# B&R Automation Studio project Panasonic_LinkaPowerCP2_A2021055 (part 21)

```iecst
			P2_Srobovanie.ServoManipulOsY.Parameters.Velocity:= P2_RemPremenne.P2_ManipSrob_OsY_Rychlost/1000;
			P2_Srobovanie.ServoManipulOsY.Parameters.Position:= P2_RemPremenne.P2_Srob_PozY_OdobratSkrutkyM4; //mm

			IF NOT SC_P2_Srobovanie.Switch1 AND P2_Pracovisko.STAV.SkrutkovackyZasunute THEN
				P2_Srobovanie.ServoManipulOsX.Command.MovePosition:= TRUE;
				P2_Srobovanie.ServoManipulOsY.Command.MovePosition:= TRUE;
				SC_P2_Srobovanie.Switch1:= TRUE;
			END_IF

			IF P2_Srobovanie.ServoManipulOsX.Status.InPosition AND P2_Srobovanie.ServoManipulOsY.Status.InPosition THEN
				P2_Srobovanie.ServoManipulOsX.Command.MovePosition:= FALSE;
				P2_Srobovanie.ServoManipulOsY.Command.MovePosition:= FALSE;
				P2_Srobovanie.STAV.ManipulatorNadPodavacmi:= TRUE;
				SC_P2_Srobovanie.ResetStep:= TRUE;
				SC_P2_Srobovanie.Step:= 242;
			END_IF

		242:
			SC_P2_Srobovanie.StepName:='242 - Automaticky Rezim - model 5H, kontrola skrutky M4 na vystupe podavaca';
			SC_P2_Srobovanie.IdleTime.PT:= T#200ms;
			SC_P2_Srobovanie.AlarmTime.PT:= T#10s;
			SC_P2_Srobovanie.AlarmTime.IN:= TRUE;

			IF P2_Srobovanie.SkrutSet_M4.IN.Podavac_SkrutkaNaVystupe THEN
				SC_P2_Srobovanie.ResetStep:= TRUE;
				SC_P2_Srobovanie.Step:= 244;
			ELSE
				P2_Srobovanie.CMD.PodajSkrutku_M4:= TRUE;
				SC_P2_Srobovanie.ResetStep:= TRUE;
				SC_P2_Srobovanie.Step:= 243;
			END_IF

		243:
			SC_P2_Srobovanie.StepName:='243 - Automaticky Rezim - model 5H, cakam na podanie skrutky M4';
			SC_P2_Srobovanie.IdleTime.PT:= T#200ms;
			SC_P2_Srobovanie.AlarmTime.PT:= T#10s;

			IF P2_Srobovanie.SkrutSet_M4.IN.Podavac_SkrutkaNaVystupe THEN
				SC_P2_Srobovanie.ResetStep:= TRUE;
				SC_P2_Srobovanie.Step:= 242;
			ELSIF P2_Srobovanie.SkrutSet_M4.STAV.ERROR THEN
				P2_Alarmy[237]:= TRUE;
				P2_Pracovisko.STAV.Porucha_ST4:= TRUE;
			END_IF

		244:
			SC_P2_Srobovanie.StepName:='244 - Automaticky Rezim - model 5H,vysunutie skrutkovacky pre odobratie skrutky M4 z podavaca';
			SC_P2_Srobovanie.IdleTime.PT:= T#2s;
			SC_P2_Srobovanie.AlarmTime.PT:= T#10s;

			P2_Srobovanie.ServoManipulOsZ_M4.Parameters.Velocity:= P2_RemPremenne.P2_ManipSrob_OsZ_M4_Rychlost/1000;
			P2_Srobovanie.ServoManipulOsZ_M4.Parameters.Position:= P2_RemPremenne.P2_Srob_PozZ_OdobratSkrutkyM4;

			IF NOT SC_P2_Srobovanie.Switch1 THEN
				P2_Srobovanie.ServoManipulOsZ_M4.Command.MovePosition:= TRUE;
				SC_P2_Srobovanie.Switch1:= TRUE;
			END_IF

			IF P2_Srobovanie.ServoManipulOsZ_M4.Status.InPosition THEN
				P2_Srobovanie.OUT.Skrutkovacka_M4_Prisavanie_OFF:= FALSE;
				P2_Srobovanie.OUT.Skrutkovacka_M4_Prisavanie_ON:= TRUE;
				SC_P2_Srobovanie.AlarmTime.IN:= TRUE;
			END_IF

			IF P2_Srobovanie.ServoManipulOsZ_M4.Status.InPosition AND P2_Srobovanie.IN.Skrutkovacka_M4_Vakum_OK THEN
				P2_Srobovanie.ServoManipulOsZ_M4.Command.MovePosition:= FALSE;
				SC_P2_Srobovanie.ResetStep:= TRUE;
				SC_P2_Srobovanie.Step:= 245;
			ELSIF SC_P2_Srobovanie.AlarmTime.Q THEN
				P2_Srobovanie.ServoManipulOsZ_M4.Command.MovePosition:= FALSE;
				P2_Srobovanie.OUT.Skrutkovacka_M4_Prisavanie_ON:= FALSE;
				P2_Srobovanie.OUT.Skrutkovacka_M4_Prisavanie_OFF:= TRUE;
				P2_Alarmy[237]:= TRUE;
				P2_Srobovanie.COM_OUT.Stav_PoruchaSkrutkovania:= TRUE;
				SC_P2_Srobovanie.ResetStep:= TRUE;
				SC_P2_Srobovanie.Step:= 245;
			END_IF

		245:
			SC_P2_Srobovanie.StepName:='245 - Automaticky Rezim - model 5H,zasunutie skrutkovacky po odobrati skrutky M4 z podavaca';
			SC_P2_Srobovanie.IdleTime.PT:= T#2s;
			SC_P2_Srobovanie.AlarmTime.PT:= T#30s;

			P2_Srobovanie.ServoManipulOsZ_M4.Parameters.Velocity:= P2_RemPremenne.P2_ManipSrob_OsZ_M4_Rychlost/1000;
			P2_Srobovanie.ServoManipulOsZ_M4.Parameters.Position:= 0;

			IF NOT SC_P2_Srobovanie.Switch1 THEN
				P2_Srobovanie.ServoManipulOsZ_M4.Command.MovePosition:= TRUE;
				SC_P2_Srobovanie.Switch1:= TRUE;
			END_IF

			IF EDGEPOS(P2_Srobovanie.ServoManipulOsZ_M4.Status.InPosition) THEN
				P2_Srobovanie.ServoManipulOsZ_M4.Command.MovePosition:= FALSE;
				IF P2_Srobovanie.COM_OUT.Stav_PoruchaSkrutkovania THEN
					P2_Pracovisko.STAV.Porucha_ST4:= TRUE;
				ELSE
					SC_P2_Srobovanie.ResetStep:= TRUE;
					SC_P2_Srobovanie.Step:= 246;
				END_IF
			END_IF

		246:
			SC_P2_Srobovanie.StepName:='246 - Automaticky Rezim - model 5H,priprava skrutky M4';
			SC_P2_Srobovanie.IdleTime.PT:= T#200ms;
			SC_P2_Srobovanie.AlarmTime.PT:= T#30s;

			P2_Srobovanie.CMD.PodajSkrutku_M4:= TRUE;
			SC_P2_Srobovanie.ResetStep:= TRUE;
			SC_P2_Srobovanie.Step:= 250;

		250:
			SC_P2_Srobovanie.StepName:='160 - Automaticky Rezim - model 5H, napolohovanie na poziciu skrutkovania strednej skrutky M4';
			SC_P2_Srobovanie.IdleTime.PT:= T#200ms;
			SC_P2_Srobovanie.AlarmTime.PT:= T#5s;

			P2_Robot.COM_OUT.ManipSrobovania_BezpecnaPozicia:= FALSE;

			IF NOT P2_Srobovanie.Manual THEN
				P2_Srobovanie.ServoManipulOsX.Parameters.Velocity:= P2_RemPremenne.P2_ManipSrob_OsX_Rychlost/1000; // m/s
				P2_Srobovanie.ServoManipulOsY.Parameters.Velocity:= P2_RemPremenne.P2_ManipSrob_OsY_Rychlost/1000; // m/s
			END_IF

			P2_Srobovanie.ServoManipulOsX.Parameters.Position:= P2_RemPremenne.P2_Srob5H_PozX_SkrutkyM4; //mm
			P2_Srobovanie.ServoManipulOsY.Parameters.Position:= P2_RemPremenne.P2_Srob5H_PozY_SkrutkyM4; //mm

			IF NOT SC_P2_Srobovanie.Switch1 AND P2_Pracovisko.STAV.SkrutkovackyZasunute THEN
				P2_Srobovanie.ServoManipulOsX.Command.MovePosition:= TRUE;
				P2_Srobovanie.ServoManipulOsY.Command.MovePosition:= TRUE;
				P2_Srobovanie.STAV.ManipulatorNadPodavacmi:= FALSE;
				SC_P2_Srobovanie.Switch1:= TRUE;
			END_IF

			IF P2_Srobovanie.ServoManipulOsX.Status.InPosition AND P2_Srobovanie.ServoManipulOsY.Status.InPosition THEN
				P2_Srobovanie.ServoManipulOsX.Command.MovePosition:= FALSE;
				P2_Srobovanie.ServoManipulOsY.Command.MovePosition:= FALSE;
				IF P2_Srobovanie.STAV.RR_Polohovanie_BUSY THEN
					P2_Srobovanie.STAV.RR_Polohovanie_BUSY:= FALSE;
					SC_P2_Srobovanie.ResetStep:= TRUE;
					SC_P2_Srobovanie.Step:= 700;
				ELSE
					SC_P2_Srobovanie.ResetStep:= TRUE;
					SC_P2_Srobovanie.Step:= 251;
				END_IF
			END_IF

		251:
			SC_P2_Srobovanie.StepName:='251 - Automaticky Rezim - model 5H, vymazanie vysledkov srobovania';
			SC_P2_Srobovanie.IdleTime.PT:= T#2s;
			SC_P2_Srobovanie.AlarmTime.PT:= T#5s;

			IF NOT SC_P2_Srobovanie.Switch1 THEN
				P2_Srobovanie.Skrutkovacka_M4.RESET_Vysledkov:= TRUE;
				SC_P2_Srobovanie.Switch1:= TRUE;
			END_IF

			IF NOT P2_Srobovanie.Skrutkovacka_M4.Stav_VysledokUtahovania_NG AND NOT P2_Srobovanie.Skrutkovacka_M4.Stav_VysledokUtahovania_OK AND NOT P2_Srobovanie.Skrutkovacka_M4.Stav_UtahovanieUkoncene THEN
				P2_Srobovanie.Skrutkovacka_M4.RESET_Vysledkov:= FALSE;
				SC_P2_Srobovanie.ResetStep:= TRUE;
				SC_P2_Srobovanie.Step:= 252;
			END_IF

		252:
			SC_P2_Srobovanie.StepName:='252 - Automaticky Rezim - model 5H, kontrola skrutkovacky a skrutky M4 v skrutkovacke';
			SC_P2_Srobovanie.IdleTime.PT:= T#2s;
			SC_P2_Srobovanie.AlarmTime.PT:= T#5s;

			IF P2_Srobovanie.IN.Skrutkovacka_M4_Vakum_OK AND P2_Srobovanie.Skrutkovacka_M4.Stav_READY_to_START THEN
				SC_P2_Srobovanie.ResetStep:= TRUE;
				SC_P2_Srobovanie.Step:= 253;
			ELSIF NOT P2_Srobovanie.Skrutkovacka_M4.Stav_READY_to_START THEN
				P2_Alarmy[275]:= TRUE;
				P2_Pracovisko.STAV.Porucha_ST4:= TRUE;
			ELSIF NOT P2_Srobovanie.IN.Skrutkovacka_M4_Vakum_OK THEN
				P2_Alarmy[237]:= TRUE;
				P2_Pracovisko.STAV.Porucha_ST4:= TRUE;
			END_IF

		253:
			SC_P2_Srobovanie.StepName:='253 - Automaticky Rezim - model 5H, vysunutie skrutkovacky M4 na poziciu pred skrutkovanim a spustenie skrutkovania';
			SC_P2_Srobovanie.IdleTime.PT:= T#500ms;
			SC_P2_Srobovanie.AlarmTime.PT:= T#10s;

			P2_Srobovanie.ServoManipulOsZ_M4.Parameters.Velocity:= P2_RemPremenne.P2_ManipSrob_OsZ_M4_Rychlost/1000;
			P2_Srobovanie.ServoManipulOsZ_M4.Parameters.Position:= 70;

			IF NOT SC_P2_Srobovanie.Switch1 THEN
				P2_Srobovanie.ServoManipulOsZ_M4.Command.MovePosition:= TRUE;
				P2_Srobovanie.Skrutkovacka_M4.START_Utahovania:= TRUE;
				P2_StoperSrobovania.STAV.VyrobaZacala:= TRUE;
				SC_P2_Srobovanie.Switch1:= TRUE;
			END_IF

			IF EDGEPOS(P2_Srobovanie.ServoManipulOsZ_M4.Status.InPosition) THEN
				P2_Srobovanie.ServoManipulOsZ_M4.Command.MovePosition:= FALSE;
				SC_P2_Srobovanie.ResetStep:= TRUE;
				SC_P2_Srobovanie.Step:= 254;
			END_IF

		254:
			SC_P2_Srobovanie.StepName:='254 - Automaticky Rezim - model 5H, prepnutie vysunutie skrutkovacky M4 na momentovy pohyb';
			SC_P2_Srobovanie.IdleTime.PT:= T#500ms;
			SC_P2_Srobovanie.AlarmTime.PT:= T#10s;
			SC_P2_Srobovanie.IdleTime.IN:= TRUE;

			P2_Srobovanie.ServoManipulOsZ_M4.Parameters.Velocity:= P2_RemPremenne.P2_Srob5H_Rychl_SkrutkyM4/1000;
			P2_Srobovanie.ServoManipulOsZ_M4.Parameters.Torque:= P2_RemPremenne.P2_Srob5H_Mom_SkrutkyM4;
			P2_Srobovanie.ServoManipulOsZ_M4.Parameters.Position:= 100;

			IF NOT SC_P2_Srobovanie.Switch1 THEN
				P2_Srobovanie.ServoManipulOsZ_M4.Command.MovePosition:= TRUE;
				SC_P2_Srobovanie.Switch1:= TRUE;
			END_IF

			IF EDGEPOS(P2_Srobovanie.ServoManipulOsZ_M4.Status.InTorque) THEN
				SC_P2_Srobovanie.ResetStep:= TRUE;
				SC_P2_Srobovanie.Step:= 255;
			END_IF

		255:
			SC_P2_Srobovanie.StepName:='255 - Automaticky Rezim - model 45F, cakam na ukoncenie skrutkovania skrutkovacky M4';
			SC_P2_Srobovanie.IdleTime.PT:= T#30s;
			SC_P2_Srobovanie.AlarmTime.PT:= T#10s;
			SC_P2_Srobovanie.IdleTime.IN:= TRUE;
			SC_P2_Srobovanie.AlarmTime.IN:= TRUE;

			IF P2_Srobovanie.Skrutkovacka_M4.Stav_UtahovanieUkoncene THEN
				P2_Srobovanie.Skrutkovacka_M4.START_Utahovania:= FALSE;
				P2_Srobovanie.ServoManipulOsZ_M4.Command.MovePosition:= FALSE;
				CasSrobovania:= TIME_TO_REAL(SC_P2_Srobovanie.IdleTime.ET);
				Reports.Skrutkovacky.VyskaSkrutkovania.P2_StrednaSkrutkaM4:= REAL_TO_STRING(P2_Srobovanie.ServoManipulOsZ_M4.Status.ActPosition);
				Reports.Skrutkovacky.CasSkrutkovania.P2_StrednaSkrutkaM4:= REAL_TO_STRING(CasSrobovania/1000);
				SC_P2_Srobovanie.ResetStep:= TRUE;
				SC_P2_Srobovanie.Step:= 256;
			ELSIF SC_P2_Srobovanie.AlarmTime.Q THEN
				P2_Alarmy[272]:= TRUE;
				CasSrobovania:= TIME_TO_REAL(SC_P2_Srobovanie.IdleTime.ET);
				Reports.Skrutkovacky.VyskaSkrutkovania.P2_StrednaSkrutkaM4:= REAL_TO_STRING(P2_Srobovanie.ServoManipulOsZ_M4.Status.ActPosition);
				Reports.Skrutkovacky.CasSkrutkovania.P2_StrednaSkrutkaM4:= REAL_TO_STRING(CasSrobovania/1000);
				P2_Srobovanie.Skrutkovacka_M4.START_Utahovania:= FALSE;
				P2_Srobovanie.COM_OUT.Stav_PoruchaSkrutkovania:= TRUE;
				P2_Srobovanie.ServoManipulOsZ_M4.Command.MovePosition:= FALSE;
				SC_P2_Srobovanie.ResetStep:= TRUE;
				SC_P2_Srobovanie.Step:= 256;
			END_IF

		256:
			SC_P2_Srobovanie.StepName:='256 - Automaticky Rezim - model 5H, zasunutie skrutkovacky M4 a vypnutie prisavania skrutky';
			SC_P2_Srobovanie.IdleTime.PT:= T#200ms;
			SC_P2_Srobovanie.AlarmTime.PT:= T#5s;

			P2_Srobovanie.ServoManipulOsZ_M4.Parameters.Velocity:= P2_RemPremenne.P2_ManipSrob_OsZ_M4_Rychlost;
			P2_Srobovanie.ServoManipulOsZ_M4.Parameters.Torque:= 1.0;
			P2_Srobovanie.ServoManipulOsZ_M4.Parameters.Position:= 0;

			IF NOT SC_P2_Srobovanie.Switch1 THEN
				P2_Srobovanie.ServoManipulOsZ_M4.Command.MovePosition:= TRUE;
				P2_Srobovanie.OUT.Skrutkovacka_M4_Prisavanie_ON:= FALSE;
				P2_Srobovanie.OUT.Skrutkovacka_M4_Prisavanie_OFF:= TRUE;
				SC_P2_Srobovanie.Switch1:= TRUE;
			END_IF

			IF EDGEPOS(P2_Srobovanie.ServoManipulOsZ_M4.Status.InPosition) THEN
				P2_Srobovanie.ServoManipulOsZ_M4.Command.MovePosition:= FALSE;
				SC_P2_Srobovanie.ResetStep:= TRUE;
				SC_P2_Srobovanie.Step:= 257;
			END_IF

		257:
			SC_P2_Srobovanie.StepName:='257 - Automaticky Rezim - model 5H, kontrola vysledkov skrutkovania strednej skrutky M4';
			SC_P2_Srobovanie.IdleTime.PT:= T#200ms;
			SC_P2_Srobovanie.AlarmTime.PT:= T#5s;

			IF P2_Srobovanie.COM_OUT.Stav_PoruchaSkrutkovania THEN
				P2_Srobovanie.STAV.Vysledok_Srobovania:= 'NG';
				P2_Srobovanie.COM_OUT.Stav_SkrutkovanieUkoncene:= TRUE;
				SC_P2_Srobovanie.ResetStep:= TRUE;
				SC_P2_Srobovanie.Step:= 258;
			ELSIF P2_Srobovanie.Skrutkovacka_M4.Stav_VysledokUtahovania_OK THEN
				P2_Srobovanie.STAV.Vysledok_Srobovania:= 'OK';
				P2_Srobovanie.COM_OUT.Stav_SkrutkovanieUkoncene:= TRUE;
				SC_P2_Srobovanie.ResetStep:= TRUE;
				SC_P2_Srobovanie.Step:= 258;
			ELSIF P2_Srobovanie.Skrutkovacka_M4.Stav_VysledokUtahovania_NG THEN
				P2_Srobovanie.STAV.Vysledok_Srobovania:= 'NG';
				P2_Srobovanie.COM_OUT.Stav_SkrutkovanieUkoncene:= TRUE;
				SC_P2_Srobovanie.ResetStep:= TRUE;
				SC_P2_Srobovanie.Step:= 258;
			END_IF

		258:
			SC_P2_Srobovanie.StepName:='258 - Automaticky Rezim - model 5H, cakam na zrusenie signalu zaskrutkuj strednu skrutku M4';
			SC_P2_Srobovanie.IdleTime.PT:= T#200ms;
			SC_P2_Srobovanie.AlarmTime.PT:= T#5s;

			IF NOT P2_Srobovanie.COM_IN.Model5H_ZaskrutkujStrednuM4 THEN
				P2_Srobovanie.COM_OUT.Stav_SkrutkovanieUkoncene:= FALSE;
				SC_P2_Srobovanie.ResetStep:= TRUE;
				SC_P2_Srobovanie.Step:= 100;
			END_IF

			//Presun manipulátora do pozície VPRED//

		400:
			SC_P2_Srobovanie.StepName:='400 - Automaticky Rezim - napolohovanie manipulatora na prednu poziciu ';
			SC_P2_Srobovanie.IdleTime.PT:= T#200ms;
			SC_P2_Srobovanie.AlarmTime.PT:= T#5s;

			P2_Robot.COM_OUT.ManipSrobovania_BezpecnaPozicia:= FALSE;

			P2_Srobovanie.ServoManipulOsX.Parameters.Velocity:= P2_RemPremenne.P2_ManipSrob_OsX_Rychlost/1000; // m/s
			P2_Srobovanie.ServoManipulOsX.Parameters.Position:= 12.5; //mm

			P2_Srobovanie.ServoManipulOsY.Parameters.Velocity:= P2_RemPremenne.P2_ManipSrob_OsY_Rychlost/1000; // m/s
			P2_Srobovanie.ServoManipulOsY.Parameters.Position:= 375; //mm

			IF NOT SC_P2_Srobovanie.Switch1 AND P2_Pracovisko.STAV.SkrutkovackyZasunute THEN
				P2_Srobovanie.ServoManipulOsY.Command.MovePosition:= TRUE;
				SC_P2_Srobovanie.Switch1:= TRUE;
			END_IF

			IF P2_Srobovanie.ServoManipulOsY.Status.ActPosition > 280 THEN
				P2_Srobovanie.ServoManipulOsX.Command.MovePosition:= TRUE;
			END_IF

			IF P2_Srobovanie.ServoManipulOsX.Status.InPosition AND P2_Srobovanie.ServoManipulOsY.Status.InPosition THEN
				P2_Srobovanie.ServoManipulOsX.Command.MovePosition:= FALSE;
				P2_Srobovanie.ServoManipulOsY.Command.MovePosition:= FALSE;
				P2_Srobovanie.COM_OUT.Stav_PresunManipulUkonceny:= TRUE;
				SC_P2_Srobovanie.ResetStep:= TRUE;
				SC_P2_Srobovanie.Step:= 402;
			END_IF

		402:
			SC_P2_Srobovanie.StepName:='402 - Automaticky Rezim - cakam na zrusenie signalu presun manipulatora vpred';
			SC_P2_Srobovanie.IdleTime.PT:= T#200ms;
			SC_P2_Srobovanie.AlarmTime.PT:= T#5s;

			IF NOT P2_Srobovanie.COM_IN.PresunManipulatora_VPRED THEN
				P2_Srobovanie.COM_OUT.Stav_PresunManipulUkonceny:= FALSE;
				SC_P2_Srobovanie.ResetStep:= TRUE;
				SC_P2_Srobovanie.Step:= 100;
			END_IF

			//Presun manipulátora do pozície VZAD//

		420:
			SC_P2_Srobovanie.StepName:='420 - Automaticky Rezim - napolohovanie manipulatora na zadnu poziciu ';
			SC_P2_Srobovanie.IdleTime.PT:= T#200ms;
			SC_P2_Srobovanie.AlarmTime.PT:= T#5s;

			P2_Robot.COM_OUT.ManipSrobovania_BezpecnaPozicia:= FALSE;

			P2_Srobovanie.ServoManipulOsX.Parameters.Velocity:= P2_RemPremenne.P2_ManipSrob_OsX_Rychlost/1000; // m/s
			P2_Srobovanie.ServoManipulOsX.Parameters.Position:= 12.5; //mm

			P2_Srobovanie.ServoManipulOsY.Parameters.Velocity:= P2_RemPremenne.P2_ManipSrob_OsY_Rychlost/1000; // m/s
			P2_Srobovanie.ServoManipulOsY.Parameters.Position:= 4.5; //mm

			IF NOT SC_P2_Srobovanie.Switch1 AND P2_Pracovisko.STAV.SkrutkovackyZasunute THEN
				P2_Srobovanie.ServoManipulOsX.Command.MovePosition:= TRUE;
				P2_Srobovanie.ServoManipulOsY.Command.MovePosition:= TRUE;
				SC_P2_Srobovanie.Switch1:= TRUE;
			END_IF

			IF P2_Srobovanie.ServoManipulOsX.Status.InPosition AND P2_Srobovanie.ServoManipulOsY.Status.InPosition THEN
				P2_Srobovanie.ServoManipulOsX.Command.MovePosition:= FALSE;
				P2_Srobovanie.ServoManipulOsY.Command.MovePosition:= FALSE;
				P2_Srobovanie.COM_OUT.Stav_PresunManipulUkonceny:= TRUE;
				SC_P2_Srobovanie.ResetStep:= TRUE;
				SC_P2_Srobovanie.Step:= 422;
			END_IF

		422:
			SC_P2_Srobovanie.StepName:='422 - Automaticky Rezim - cakam na zrusenie signalu presun manipulatora vzad';
			SC_P2_Srobovanie.IdleTime.PT:= T#200ms;
			SC_P2_Srobovanie.AlarmTime.PT:= T#5s;

			IF NOT P2_Srobovanie.COM_IN.PresunManipulatora_VZAD THEN
				P2_Srobovanie.COM_OUT.Stav_PresunManipulUkonceny:= FALSE;
				SC_P2_Srobovanie.ResetStep:= TRUE;
				SC_P2_Srobovanie.Step:= 100;
			END_IF

			//Odobratie skrutky M4//
		440:
			SC_P2_Srobovanie.StepName:='440 - Automaticky Rezim - odobratie skrtuky M4, napolohovanie zadnej skrutkovacky M4 na poziciu odobratia skrutky M4 z podavaca';
			SC_P2_Srobovanie.IdleTime.PT:= T#200ms;
			SC_P2_Srobovanie.AlarmTime.PT:= T#5s;

			P2_Robot.COM_OUT.ManipSrobovania_BezpecnaPozicia:= FALSE;

			IF NOT P2_Srobovanie.Manual THEN
				P2_Srobovanie.ServoManipulOsX.Parameters.Velocity:= P2_RemPremenne.P2_ManipSrob_OsX_Rychlost/1000; // m/s
				P2_Srobovanie.ServoManipulOsY.Parameters.Velocity:= P2_RemPremenne.P2_ManipSrob_OsY_Rychlost/1000; // m/s
			END_IF

			P2_Srobovanie.ServoManipulOsX.Parameters.Position:= P2_RemPremenne.P2_Srob_PozX_OdobratSkrutkyM4; //mm
			P2_Srobovanie.ServoManipulOsY.Parameters.Position:= P2_RemPremenne.P2_Srob_PozY_OdobratSkrutkyM4; //mm

			IF NOT SC_P2_Srobovanie.Switch1 AND P2_Pracovisko.STAV.SkrutkovackyZasunute THEN
				P2_Srobovanie.ServoManipulOsX.Command.MovePosition:= TRUE;
				P2_Srobovanie.ServoManipulOsY.Command.MovePosition:= TRUE;
				SC_P2_Srobovanie.Switch1:= TRUE;
			END_IF

			IF P2_Srobovanie.ServoManipulOsX.Status.InPosition AND P2_Srobovanie.ServoManipulOsY.Status.InPosition THEN
				P2_Srobovanie.ServoManipulOsX.Command.MovePosition:= FALSE;
				P2_Srobovanie.ServoManipulOsY.Command.MovePosition:= FALSE;
				P2_Srobovanie.STAV.ManipulatorNadPodavacmi:= TRUE;
				IF P2_Srobovanie.STAV.RR_Polohovanie_BUSY THEN
					P2_Srobovanie.STAV.RR_Polohovanie_BUSY:= FALSE;
					SC_P2_Srobovanie.ResetStep:= TRUE;
					SC_P2_Srobovanie.Step:= 700;
				ELSE
					SC_P2_Srobovanie.ResetStep:= TRUE;
					SC_P2_Srobovanie.Step:= 442;
				END_IF
			END_IF

		442:
			SC_P2_Srobovanie.StepName:='442 - Automaticky Rezim - odobratie skrutky M4, kontrola skrutky M4 na vystupe podavaca';
			SC_P2_Srobovanie.IdleTime.PT:= T#200ms;
			SC_P2_Srobovanie.AlarmTime.PT:= T#10s;
			SC_P2_Srobovanie.AlarmTime.IN:= TRUE;

			IF P2_Srobovanie.IN.Skrutkovacka_M4_Vakum_OK THEN
				SC_P2_Srobovanie.ResetStep:= TRUE;
				SC_P2_Srobovanie.Step:= 450;
			ELSIF P2_Srobovanie.SkrutSet_M4.IN.Podavac_SkrutkaNaVystupe THEN
				SC_P2_Srobovanie.ResetStep:= TRUE;
				SC_P2_Srobovanie.Step:= 447;
			ELSIF NOT P2_Srobovanie.SkrutSet_M4.IN.Podavac_SkrutkaNaVystupe THEN
				P2_Srobovanie.CMD.PodajSkrutku_M4:= TRUE;
				SC_P2_Srobovanie.ResetStep:= TRUE;
				SC_P2_Srobovanie.Step:= 445;
			END_IF

		445:
			SC_P2_Srobovanie.StepName:='445 - Automaticky Rezim - odobratie skrutky M4, cakam na podanie skrutky M4';
			SC_P2_Srobovanie.IdleTime.PT:= T#200ms;
			SC_P2_Srobovanie.AlarmTime.PT:= T#10s;

			IF P2_Srobovanie.SkrutSet_M4.IN.Podavac_SkrutkaNaVystupe THEN
				SC_P2_Srobovanie.ResetStep:= TRUE;
				SC_P2_Srobovanie.Step:= 442;
			ELSIF P2_Srobovanie.SkrutSet_M4.STAV.ERROR THEN
				P2_Alarmy[237]:= TRUE;
				P2_Pracovisko.STAV.Porucha_ST4:= TRUE;
			END_IF

		447:
			SC_P2_Srobovanie.StepName:='447 - Automaticky Rezim - odobratie skrutky M4,vysunutie skrutkovacky pre odobratie skrutky M4 z podavaca';
			SC_P2_Srobovanie.IdleTime.PT:= T#2s;
			SC_P2_Srobovanie.AlarmTime.PT:= T#10s;

			P2_Srobovanie.ServoManipulOsZ_M4.Parameters.Velocity:= P2_RemPremenne.P2_ManipSrob_OsZ_M4_Rychlost/1000;
			P2_Srobovanie.ServoManipulOsZ_M4.Parameters.Position:= P2_RemPremenne.P2_Srob_PozZ_OdobratSkrutkyM4;

			IF NOT SC_P2_Srobovanie.Switch1 THEN
				P2_Srobovanie.ServoManipulOsZ_M4.Command.MovePosition:= TRUE;
				SC_P2_Srobovanie.Switch1:= TRUE;
			END_IF

			IF P2_Srobovanie.ServoManipulOsZ_M4.Status.InPosition THEN
				P2_Srobovanie.OUT.Skrutkovacka_M4_Prisavanie_OFF:= FALSE;
				P2_Srobovanie.OUT.Skrutkovacka_M4_Prisavanie_ON:= TRUE;
				SC_P2_Srobovanie.AlarmTime.IN:= TRUE;
			END_IF

			IF P2_Srobovanie.ServoManipulOsZ_M4.Status.InPosition AND P2_Srobovanie.IN.Skrutkovacka_M4_Vakum_OK THEN
				P2_Srobovanie.ServoManipulOsZ_M4.Command.MovePosition:= FALSE;
				SC_P2_Srobovanie.ResetStep:= TRUE;
				SC_P2_Srobovanie.Step:= 448;
			ELSIF SC_P2_Srobovanie.AlarmTime.Q THEN
				P2_Srobovanie.ServoManipulOsZ_M4.Command.MovePosition:= FALSE;
				P2_Srobovanie.OUT.Skrutkovacka_M4_Prisavanie_ON:= FALSE;
				P2_Srobovanie.OUT.Skrutkovacka_M4_Prisavanie_OFF:= TRUE;
				P2_Alarmy[237]:= TRUE;
				P2_Srobovanie.COM_OUT.Stav_PoruchaSkrutkovania:= TRUE;
				SC_P2_Srobovanie.ResetStep:= TRUE;
				SC_P2_Srobovanie.Step:= 448;
			END_IF

		448:
			SC_P2_Srobovanie.StepName:='448 - Automaticky Rezim - odobratie skrutky M4,zasunutie skrutkovacky po odobrati skrutky M4 z podavaca';
			SC_P2_Srobovanie.IdleTime.PT:= T#2s;
			SC_P2_Srobovanie.AlarmTime.PT:= T#30s;

			P2_Srobovanie.ServoManipulOsZ_M4.Parameters.Velocity:= P2_RemPremenne.P2_ManipSrob_OsZ_M4_Rychlost/1000;
			P2_Srobovanie.ServoManipulOsZ_M4.Parameters.Position:= 0;

			IF NOT SC_P2_Srobovanie.Switch1 THEN
				P2_Srobovanie.ServoManipulOsZ_M4.Command.MovePosition:= TRUE;
				SC_P2_Srobovanie.Switch1:= TRUE;
			END_IF

			IF EDGEPOS(P2_Srobovanie.ServoManipulOsZ_M4.Status.InPosition) THEN
				P2_Srobovanie.ServoManipulOsZ_M4.Command.MovePosition:= FALSE;
				IF P2_Srobovanie.COM_OUT.Stav_PoruchaSkrutkovania THEN
					P2_Pracovisko.STAV.Porucha_ST4:= TRUE;
				ELSE
					SC_P2_Srobovanie.ResetStep:= TRUE;
					SC_P2_Srobovanie.Step:= 450;
				END_IF
			END_IF

		450:
			SC_P2_Srobovanie.StepName:='450 - Automaticky Rezim - odobratie skrutky M4,priprava skrutky M4';
			SC_P2_Srobovanie.IdleTime.PT:= T#200ms;
			SC_P2_Srobovanie.AlarmTime.PT:= T#30s;

			P2_Srobovanie.CMD.PodajSkrutku_M4:= TRUE;
			SC_P2_Srobovanie.ResetStep:= TRUE;
			SC_P2_Srobovanie.Step:= 455;

		455:
			SC_P2_Srobovanie.StepName:='455 - Automaticky Rezim - odobratie skrutky M4, cakam na zrusenie signalu odober skrutku M4';
			SC_P2_Srobovanie.IdleTime.PT:= T#200ms;
			SC_P2_Srobovanie.AlarmTime.PT:= T#5s;

			P2_Srobovanie.COM_OUT.Stav_SkrutkovanieUkoncene:= TRUE;

			IF NOT P2_Srobovanie.COM_IN.OdoberSkrutku_M4 THEN
				P2_Srobovanie.COM_OUT.Stav_SkrutkovanieUkoncene:= FALSE;
				P2_Srobovanie.STAV.ManipulatorNadPodavacmi:= FALSE;
				SC_P2_Srobovanie.ResetStep:= TRUE;
				SC_P2_Srobovanie.Step:= 100;
			END_IF

			//*********************************************************Čistenie skrutkovačiek*****************************************************************************//

			//Čistenie skrutkovačky M5//
		500:
			SC_P2_Srobovanie.StepName:='500 - Automaticky Rezim - cistenie skrutkovacky M5,kontrola zrusenia stavu serva v pozicii';
			SC_P2_Srobovanie.IdleTime.PT:= T#300ms;
			SC_P2_Srobovanie.AlarmTime.PT:= T#5s;

			P2_Srobovanie.STAV.CistenieSkrutkovackyM5_BUSY:= TRUE;
			P2_Srobovanie.STAV.SkrutkaM5_READY:= FALSE;

			IF NOT P2_Srobovanie.ServoManipulOsX.Status.InPosition AND NOT P2_Srobovanie.ServoManipulOsY.Status.InPosition THEN
				SC_P2_Srobovanie.ResetStep:= TRUE;
				SC_P2_Srobovanie.Step:= 501;
			END_IF

		501:
			SC_P2_Srobovanie.StepName:='501 - Automaticky Rezim - cistenie skrutkovacky M5,presun na poziciu zahodenia skrutky';
			SC_P2_Srobovanie.IdleTime.PT:= T#300ms;
			SC_P2_Srobovanie.AlarmTime.PT:= T#5s;

			P2_Robot.COM_OUT.ManipSrobovania_BezpecnaPozicia:= FALSE;

			IF NOT P2_Srobovanie.Manual THEN
				P2_Srobovanie.ServoManipulOsX.Parameters.Velocity:= P2_RemPremenne.P2_ManipSrob_OsX_Rychlost/1000; // m/s
				P2_Srobovanie.ServoManipulOsY.Parameters.Velocity:= P2_RemPremenne.P2_ManipSrob_OsY_Rychlost/1000; // m/s
			END_IF

			P2_Srobovanie.ServoManipulOsX.Parameters.Position:= 35; //mm
			P2_Srobovanie.ServoManipulOsY.Parameters.Position:= 85; //mm

			IF NOT SC_P2_Srobovanie.Switch1 AND P2_Pracovisko.STAV.SkrutkovackyZasunute THEN
				P2_Srobovanie.ServoManipulOsX.Command.MovePosition:= TRUE;
				P2_Srobovanie.ServoManipulOsY.Command.MovePosition:= TRUE;
				SC_P2_Srobovanie.Switch1:= TRUE;
			END_IF

			IF P2_Srobovanie.ServoManipulOsX.Status.InPosition AND P2_Srobovanie.ServoManipulOsY.Status.InPosition THEN
				P2_Srobovanie.ServoManipulOsX.Command.MovePosition:= FALSE;
				P2_Srobovanie.ServoManipulOsY.Command.MovePosition:= FALSE;
				SC_P2_Srobovanie.ResetStep:= TRUE;
				SC_P2_Srobovanie.Step:= 502;
			END_IF

		502:
			SC_P2_Srobovanie.StepName:='502 - Automaticky Rezim - cistenie skrutkovacky M5,vysunutie skrutkovacky M5';
			SC_P2_Srobovanie.IdleTime.PT:= T#1s;
			SC_P2_Srobovanie.AlarmTime.PT:= T#2s;

			IF NOT SC_P2_Srobovanie.Switch1 THEN
				P2_Srobovanie.OUT.Skrutkovacka_M5_Prisavanie_ON:= TRUE;
				P2_Srobovanie.OUT.Skrutkovacku_M5_VYSUN:= TRUE;
				SC_P2_Srobovanie.IdleTime.IN:= TRUE;
				SC_P2_Srobovanie.Switch1:= TRUE;
			END_IF

			IF SC_P2_Srobovanie.IdleTime.Q THEN
				P2_Srobovanie.OUT.Skrutkovacka_M5_Prisavanie_ON:= FALSE;
				SC_P2_Srobovanie.AlarmTime.IN:= TRUE;
			END_IF

			IF SC_P2_Srobovanie.AlarmTime.Q THEN
				P2_Srobovanie.OUT.Skrutkovacku_M5_VYSUN:= FALSE;
				SC_P2_Srobovanie.ResetStep:= TRUE;
				SC_P2_Srobovanie.Step:= 505;
			END_IF

		505:
			SC_P2_Srobovanie.StepName:='505 - Automaticky Rezim - cistenie skrutkovacky M5,nabitie skrutky do skrutkovacky M5';
			SC_P2_Srobovanie.IdleTime.PT:= T#2s;
			SC_P2_Srobovanie.AlarmTime.PT:= T#30s;

			IF NOT SC_P2_Srobovanie.Switch1 AND P2_Srobovanie.IN.Skrutkovacka_M5_ZASUNUTA THEN
				IF P2_Srobovanie.Manual THEN
					P2_Srobovanie.CMD.RR_SkrutSetM5_PodajSkrutku:= TRUE;
				ELSE
					P2_Srobovanie.CMD.PodajSkrutku_M5:= TRUE;
				END_IF
				SC_P2_Srobovanie.Switch1:= TRUE;
			END_IF

			IF P2_Srobovanie.STAV.SkrutkaM5_READY THEN
				P2_Srobovanie.STAV.CistenieSkrutkovackyM5_BUSY:= FALSE;
				SC_P2_Srobovanie.ResetStep:= TRUE;
				SC_P2_Srobovanie.Step:= FazaNavratu;
			ELSIF P2_Srobovanie.SkrutSet_M5.Error.ErrorBit THEN
				P2_Alarmy[238]:= TRUE;
				P2_Pracovisko.STAV.Porucha_ST4:= TRUE;
			END_IF

			//Čistenie skrutkovačky M4//
		520:
			SC_P2_Srobovanie.StepName:='520 - Automaticky Rezim - cistenie skrutkovacky M4,kontrola zrusenia stavu serva v pozicii';
			SC_P2_Srobovanie.IdleTime.PT:= T#300ms;
			SC_P2_Srobovanie.AlarmTime.PT:= T#5s;

			IF NOT P2_Srobovanie.ServoManipulOsX.Status.InPosition AND NOT P2_Srobovanie.ServoManipulOsY.Status.InPosition THEN
				SC_P2_Srobovanie.ResetStep:= TRUE;
				SC_P2_Srobovanie.Step:= 521;
			END_IF

		521:
			SC_P2_Srobovanie.StepName:='521 - Automaticky Rezim - cistenie skrutkovacky M4,presun manipulatora na poziciu zahodenia skrutky M4';
			SC_P2_Srobovanie.IdleTime.PT:= T#300ms;
			SC_P2_Srobovanie.AlarmTime.PT:= T#5s;

			P2_Robot.COM_OUT.ManipSrobovania_BezpecnaPozicia:= FALSE;

			IF NOT P2_Srobovanie.Manual THEN
				P2_Srobovanie.ServoManipulOsX.Parameters.Velocity:= P2_RemPremenne.P2_ManipSrob_OsX_Rychlost/1000; // m/s
				P2_Srobovanie.ServoManipulOsY.Parameters.Velocity:= P2_RemPremenne.P2_ManipSrob_OsY_Rychlost/1000; // m/s
			END_IF

			P2_Srobovanie.ServoManipulOsX.Parameters.Position:= 23; //mm
			P2_Srobovanie.ServoManipulOsY.Parameters.Position:= 150; //mm

			IF NOT SC_P2_Srobovanie.Switch1 AND P2_Pracovisko.STAV.SkrutkovackyZasunute THEN
				P2_Srobovanie.ServoManipulOsX.Command.MovePosition:= TRUE;
				P2_Srobovanie.ServoManipulOsY.Command.MovePosition:= TRUE;
				SC_P2_Srobovanie.Switch1:= TRUE;
			END_IF

			IF P2_Srobovanie.ServoManipulOsX.Status.InPosition AND P2_Srobovanie.ServoManipulOsY.Status.InPosition THEN
				P2_Srobovanie.ServoManipulOsX.Command.MovePosition:= FALSE;
				P2_Srobovanie.ServoManipulOsY.Command.MovePosition:= FALSE;
				SC_P2_Srobovanie.ResetStep:= TRUE;
				SC_P2_Srobovanie.Step:= 523;
			END_IF

		523:
			SC_P2_Srobovanie.StepName:='523 - Automaticky Rezim - cistenie skrutkovacky M4, vysuvam skrutkovac M4 a vypinam prisavanie skrutky,priprava skrutky M4';
			SC_P2_Srobovanie.IdleTime.PT:= T#2s;
			SC_P2_Srobovanie.AlarmTime.PT:= T#30s;

			P2_Srobovanie.ServoManipulOsZ_M4.Parameters.Velocity:= P2_RemPremenne.P2_ManipSrob_OsZ_M4_Rychlost/1000;
			P2_Srobovanie.ServoManipulOsZ_M4.Parameters.Position:= 99;

			IF NOT SC_P2_Srobovanie.Switch1 THEN
				P2_Srobovanie.ServoManipulOsZ_M4.Command.MovePosition:= TRUE;
				P2_Srobovanie.CMD.PodajSkrutku_M4:= TRUE;
				SC_P2_Srobovanie.Switch1:= TRUE;
			END_IF

			IF P2_Srobovanie.ServoManipulOsZ_M4.Status.InPosition THEN
				P2_Srobovanie.ServoManipulOsZ_M4.Command.MovePosition:= FALSE;
				P2_Srobovanie.OUT.Skrutkovacka_M4_Prisavanie_ON:= FALSE;
				P2_Srobovanie.OUT.Skrutkovacka_M4_Prisavanie_OFF:= TRUE;
				SC_P2_Srobovanie.ResetStep:= TRUE;
				SC_P2_Srobovanie.Step:= 525;
			END_IF

		525:
			SC_P2_Srobovanie.StepName:='525 - Automaticky Rezim - cistenie skrutkovacky M4, otretie skrutkovacky M4';
			SC_P2_Srobovanie.IdleTime.PT:= T#2s;
			SC_P2_Srobovanie.AlarmTime.PT:= T#30s;

			P2_Robot.COM_OUT.ManipSrobovania_BezpecnaPozicia:= FALSE;

			P2_Srobovanie.ServoManipulOsX.Parameters.Velocity:= P2_RemPremenne.P2_ManipSrob_OsX_Rychlost/1000;
			P2_Srobovanie.ServoManipulOsX.Parameters.Position:= 5; //mm

			P2_Srobovanie.ServoManipulOsY.Parameters.Velocity:= P2_RemPremenne.P2_ManipSrob_OsY_Rychlost/1000;
			P2_Srobovanie.ServoManipulOsY.Parameters.Position:= 150; //mm

			IF NOT SC_P2_Srobovanie.Switch1 THEN
				P2_Srobovanie.ServoManipulOsX.Command.MovePosition:= TRUE;
				P2_Srobovanie.ServoManipulOsY.Command.MovePosition:= TRUE;
				SC_P2_Srobovanie.Switch1:= TRUE;
			END_IF

			IF P2_Srobovanie.ServoManipulOsX.Status.InPosition AND P2_Srobovanie.ServoManipulOsY.Status.InPosition AND NOT P2_Srobovanie.IN.Skrutkovacka_M4_Vakum_OK THEN
				P2_Srobovanie.ServoManipulOsX.Command.MovePosition:= FALSE;
				P2_Srobovanie.ServoManipulOsY.Command.MovePosition:= FALSE;
				SC_P2_Srobovanie.ResetStep:= TRUE;
				SC_P2_Srobovanie.Step:= 528;
			END_IF

		528:
			SC_P2_Srobovanie.StepName:='528 - Automaticky Rezim - cistenie skrutkovacky M4, zasuvam skrutkovac M4';
			SC_P2_Srobovanie.IdleTime.PT:= T#2s;
			SC_P2_Srobovanie.AlarmTime.PT:= T#30s;

			P2_Srobovanie.ServoManipulOsZ_M4.Parameters.Velocity:= P2_RemPremenne.P2_ManipSrob_OsZ_M4_Rychlost/1000;
			P2_Srobovanie.ServoManipulOsZ_M4.Parameters.Position:= 0;

			IF NOT SC_P2_Srobovanie.Switch1 THEN
				P2_Srobovanie.ServoManipulOsZ_M4.Command.MovePosition:= TRUE;
				SC_P2_Srobovanie.Switch1:= TRUE;
			END_IF

			IF P2_Srobovanie.ServoManipulOsZ_M4.Status.InPosition AND P2_Srobovanie.SkrutSet_M4.IN.Podavac_SkrutkaNaVystupe AND NOT P2_Srobovanie.IN.Skrutkovacka_M4_Vakum_OK THEN
				P2_Srobovanie.ServoManipulOsZ_M4.Command.MovePosition:= FALSE;
				SC_P2_Srobovanie.ResetStep:= TRUE;
				SC_P2_Srobovanie.Step:= FazaNavratu;
			ELSIF P2_Srobovanie.SkrutSet_M4.STAV.ERROR THEN
				P2_Alarmy[237]:= TRUE;
				P2_Pracovisko.STAV.Porucha_ST4:= TRUE;
			END_IF

			//Čistenie skrutkovačky M6//
		600:
			SC_P2_Srobovanie.StepName:='600 - Automaticky Rezim - cistenie skrutkovacky M6,kontrola zrusenia stavu serva v pozicii';
			SC_P2_Srobovanie.IdleTime.PT:= T#300ms;
			SC_P2_Srobovanie.AlarmTime.PT:= T#5s;

			P2_Srobovanie.STAV.CistenieSkrutkovackyM6_BUSY:= TRUE;
			P2_Srobovanie.STAV.SkrutkaM6_READY:= FALSE;

			IF NOT P2_Srobovanie.ServoManipulOsX.Status.InPosition AND NOT P2_Srobovanie.ServoManipulOsY.Status.InPosition THEN
				SC_P2_Srobovanie.ResetStep:= TRUE;
				SC_P2_Srobovanie.Step:= 601;
			END_IF

		601:
			SC_P2_Srobovanie.StepName:='601 - Automaticky Rezim - cistenie skrutkovacky M6,presun na poziciu zahodenia skrutky';
			SC_P2_Srobovanie.IdleTime.PT:= T#300ms;
			SC_P2_Srobovanie.AlarmTime.PT:= T#5s;

			P2_Robot.COM_OUT.ManipSrobovania_BezpecnaPozicia:= FALSE;

			IF NOT P2_Srobovanie.Manual THEN
				P2_Srobovanie.ServoManipulOsX.Parameters.Velocity:= P2_RemPremenne.P2_ManipSrob_OsX_Rychlost/1000; // m/s
				P2_Srobovanie.ServoManipulOsY.Parameters.Velocity:= P2_RemPremenne.P2_ManipSrob_OsY_Rychlost/1000; // m/s
			END_IF

			P2_Srobovanie.ServoManipulOsX.Parameters.Position:= 35; //mm
			P2_Srobovanie.ServoManipulOsY.Parameters.Position:= 5; //mm

			IF NOT SC_P2_Srobovanie.Switch1 AND P2_Pracovisko.STAV.SkrutkovackyZasunute THEN
				P2_Srobovanie.ServoManipulOsX.Command.MovePosition:= TRUE;
				P2_Srobovanie.ServoManipulOsY.Command.MovePosition:= TRUE;
				SC_P2_Srobovanie.Switch1:= TRUE;
			END_IF

			IF P2_Srobovanie.ServoManipulOsX.Status.InPosition AND P2_Srobovanie.ServoManipulOsY.Status.InPosition THEN
				P2_Srobovanie.ServoManipulOsX.Command.MovePosition:= FALSE;
				P2_Srobovanie.ServoManipulOsY.Command.MovePosition:= FALSE;
				SC_P2_Srobovanie.ResetStep:= TRUE;
				SC_P2_Srobovanie.Step:= 602;
			END_IF

		602:
			SC_P2_Srobovanie.StepName:='602 - Automaticky Rezim - cistenie skrutkovacky M6,vysunutie skrutkovacky M6';
			SC_P2_Srobovanie.IdleTime.PT:= T#1s;
			SC_P2_Srobovanie.AlarmTime.PT:= T#2s;

			IF NOT SC_P2_Srobovanie.Switch1 THEN
				P2_Srobovanie.OUT.Skrutkovacka_M6_Prisavanie_ON:= TRUE;
				P2_Srobovanie.OUT.Skrutkovacku_M6_VYSUN:= TRUE;
				SC_P2_Srobovanie.IdleTime.IN:= TRUE;
				SC_P2_Srobovanie.Switch1:= TRUE;
			END_IF

			IF SC_P2_Srobovanie.IdleTime.Q THEN
				P2_Srobovanie.OUT.Skrutkovacka_M6_Prisavanie_ON:= FALSE;
				SC_P2_Srobovanie.AlarmTime.IN:= TRUE;
			END_IF

			IF SC_P2_Srobovanie.AlarmTime.Q THEN
				P2_Srobovanie.OUT.Skrutkovacku_M6_VYSUN:= FALSE;
				SC_P2_Srobovanie.ResetStep:= TRUE;
				SC_P2_Srobovanie.Step:= 605;
			END_IF

		605:
			SC_P2_Srobovanie.StepName:='605 - Automaticky Rezim - cistenie skrutkovacky M6,nabitie skrutky do skrutkovacky M6';
			SC_P2_Srobovanie.IdleTime.PT:= T#2s;
			SC_P2_Srobovanie.AlarmTime.PT:= T#30s;

			IF NOT SC_P2_Srobovanie.Switch1 AND P2_Srobovanie.IN.Skrutkovacka_M6_ZASUNUTA THEN
				IF P2_Srobovanie.Manual THEN
					P2_Srobovanie.CMD.RR_SkrutSetM6_PodajSkrutku:= TRUE;
				ELSE
					P2_Srobovanie.CMD.PodajSkrutku_M6:= TRUE;
				END_IF
				SC_P2_Srobovanie.Switch1:= TRUE;
			END_IF

			IF P2_Srobovanie.STAV.SkrutkaM6_READY THEN
				P2_Srobovanie.STAV.CistenieSkrutkovackyM6_BUSY:= FALSE;
				SC_P2_Srobovanie.ResetStep:= TRUE;
				SC_P2_Srobovanie.Step:= FazaNavratu;
			ELSIF P2_Srobovanie.SkrutSet_M6.Error.ErrorBit THEN
				P2_Alarmy[239]:= TRUE;
				P2_Pracovisko.STAV.Porucha_ST4:= TRUE;
			END_IF

			//*******************************************************Manuálny režim*******************************************************************************//
		700:
			SC_P2_Srobovanie.StepName:='700 - Manualny Rezim';
			SC_P2_Srobovanie.IdleTime.PT:= T#8s;
			SC_P2_Srobovanie.AlarmTime.PT:= T#5s;

			//Ovládanie manipulátora os X//

			P2_Srobovanie.ServoManipulOsX.Parameters.Acc:= 1;
			P2_Srobovanie.ServoManipulOsX.Parameters.Dcc:= 1;
			P2_Srobovanie.ServoManipulOsX.Parameters.Velocity:= P2_Srobovanie.PAR.ManipulOsX_JoggRychlost/1000;
			P2_Srobovanie.ServoManipulOsX.Command.TorqueLimitation:= TRUE;
			P2_Srobovanie.ServoManipulOsX.Parameters.Torque:= 1;

			IF P2_Srobovanie.CMD.RR_Manipulator_OsX_VPRAVO AND NOT P2_Srobovanie.ServoManipulOsX.Command.Stop AND P2_Pracovisko.STAV.SkrutkovackyZasunute THEN
				P2_Srobovanie.ServoManipulOsX.Parameters.Position:= 45;
				P2_Srobovanie.ServoManipulOsX.Command.MovePosition:= TRUE;
			ELSIF P2_Srobovanie.CMD.RR_Manipulator_OsX_VLAVO AND NOT P2_Srobovanie.ServoManipulOsX.Command.Stop AND P2_Pracovisko.STAV.SkrutkovackyZasunute THEN
				P2_Srobovanie.ServoManipulOsX.Parameters.Position:= 0;
				P2_Srobovanie.ServoManipulOsX.Command.MovePosition:= TRUE;
			ELSE
				P2_Srobovanie.ServoManipulOsX.Command.MovePosition:= FALSE;
				P2_Srobovanie.ServoManipulOsX.Command.Stop:= TRUE;
			END_IF

			IF P2_Srobovanie.ServoManipulOsX.Command.Stop AND P2_Srobovanie.ServoManipulOsX.Status.StandStill THEN
				P2_Srobovanie.ServoManipulOsX.Command.Stop:= FALSE;
			END_IF

			//Ovládanie manipulátora os Y//
			P2_Srobovanie.ServoManipulOsY.Parameters.Acc:= 1;
			P2_Srobovanie.ServoManipulOsY.Parameters.Dcc:= 1;
			P2_Srobovanie.ServoManipulOsY.Parameters.Velocity:= P2_Srobovanie.PAR.ManipulOsY_JoggRychlost/1000;
			P2_Srobovanie.ServoManipulOsY.Command.TorqueLimitation:= TRUE;
			P2_Srobovanie.ServoManipulOsY.Parameters.Torque:= 1;

			IF P2_Srobovanie.CMD.RR_Manipulator_OsY_VPRED AND NOT P2_Srobovanie.ServoManipulOsY.Command.Stop AND P2_Pracovisko.STAV.SkrutkovackyZasunute THEN
				P2_Srobovanie.ServoManipulOsY.Parameters.Position:= 320;
				P2_Srobovanie.ServoManipulOsY.Command.MovePosition:= TRUE;
			ELSIF P2_Srobovanie.CMD.RR_Manipulator_OsY_VZAD AND NOT P2_Srobovanie.ServoManipulOsY.Command.Stop AND P2_Pracovisko.STAV.SkrutkovackyZasunute THEN
				P2_Srobovanie.ServoManipulOsY.Parameters.Position:= 0;
				P2_Srobovanie.ServoManipulOsY.Command.MovePosition:= TRUE;
			ELSE
				P2_Srobovanie.ServoManipulOsY.Command.MovePosition:= FALSE;
				P2_Srobovanie.ServoManipulOsY.Command.Stop:= TRUE;
			END_IF

			IF P2_Srobovanie.ServoManipulOsY.Command.Stop AND P2_Srobovanie.ServoManipulOsY.Status.StandStill THEN
				P2_Srobovanie.ServoManipulOsY.Command.Stop:= FALSE;
			END_IF

			//Ovládanie vysunutia skrutkovačky M4//
			P2_Srobovanie.ServoManipulOsZ_M4.Parameters.Acc:= 1;
			P2_Srobovanie.ServoManipulOsZ_M4.Parameters.Dcc:= 1;
			P2_Srobovanie.ServoManipulOsZ_M4.Parameters.Velocity:= P2_Srobovanie.PAR.ManipulOsZ_M4_JoggRychlost/1000;
			P2_Srobovanie.ServoManipulOsZ_M4.Command.TorqueLimitation:= TRUE;
			(*P2_Srobovanie.ServoManipulOsZ_M4.Parameters.Torque:= 1;*)

			IF P2_Srobovanie.CMD.RR_SkrutkovackaM4_OsZ_DOLE AND NOT P2_Srobovanie.ServoManipulOsZ_M4.Command.Stop THEN
				P2_Srobovanie.ServoManipulOsZ_M4.Parameters.Position:= 100;
				P2_Srobovanie.ServoManipulOsZ_M4.Command.MovePosition:= TRUE;
			ELSIF P2_Srobovanie.CMD.RR_SkrutkovackaM4_OsZ_HORE AND NOT P2_Srobovanie.ServoManipulOsZ_M4.Command.Stop THEN
				P2_Srobovanie.ServoManipulOsZ_M4.Parameters.Position:= 0;
				P2_Srobovanie.ServoManipulOsZ_M4.Command.MovePosition:= TRUE;
			ELSE
				P2_Srobovanie.ServoManipulOsZ_M4.Command.MovePosition:= FALSE;
				P2_Srobovanie.ServoManipulOsZ_M4.Command.Stop:= TRUE;
			END_IF

			IF P2_Srobovanie.ServoManipulOsZ_M4.Command.Stop AND P2_Srobovanie.ServoManipulOsZ_M4.Status.StandStill THEN
				P2_Srobovanie.ServoManipulOsZ_M4.Command.Stop:= FALSE;
			END_IF

			//Prisávanie skrutky M4//
			IF P2_Srobovanie.CMD.RR_PrisavanieSkrutkyM4_ON THEN
				P2_Srobovanie.OUT.Skrutkovacka_M4_Prisavanie_OFF:= FALSE;
				P2_Srobovanie.OUT.Skrutkovacka_M4_Prisavanie_ON:= TRUE;
				P2_Srobovanie.CMD.RR_PrisavanieSkrutkyM4_ON:= FALSE;
			ELSIF P2_Srobovanie.CMD.RR_PrisavanieSkrutkyM4_OFF THEN
				P2_Srobovanie.OUT.Skrutkovacka_M4_Prisavanie_ON:= FALSE;
				P2_Srobovanie.OUT.Skrutkovacka_M4_Prisavanie_OFF:= TRUE;
				P2_Srobovanie.CMD.RR_PrisavanieSkrutkyM4_OFF:= FALSE;
			END_IF

			//Čistenie skrutkovačky M6//
			IF P2_Srobovanie.CMD.RR_CistenieSkrutkovackyM6 THEN
				IF P2_Pracovisko.STAV.SkrutkovackyZasunute AND Safety.STAV.P2_ZonaBunky_AKTIVNA THEN
					FazaNavratu:= 700;
					SC_P2_Srobovanie.ResetStep:= TRUE;
					SC_P2_Srobovanie.Step:= 600;
				END_IF
				P2_Srobovanie.CMD.RR_CistenieSkrutkovackyM6:= FALSE;
			END_IF

			//Čistenie skrutkovačky M5//
			IF P2_Srobovanie.CMD.RR_CistenieSkrutkovackyM5 THEN
				IF P2_Pracovisko.STAV.SkrutkovackyZasunute AND Safety.STAV.P2_ZonaBunky_AKTIVNA THEN
					FazaNavratu:= 700;
					SC_P2_Srobovanie.ResetStep:= TRUE;
					SC_P2_Srobovanie.Step:= 500;
				END_IF
				P2_Srobovanie.CMD.RR_CistenieSkrutkovackyM5:= FALSE;
			END_IF

			//**********************Polohovanie na pozície skrutiek*****************************//
			IF P2_Srobovanie.CMD.RR_PolohujManipulator THEN
				IF P2_Pracovisko.STAV.SkrutkovackyZasunute THEN
					IF P2_Srobovanie.PAR.RR_IndexPolohovaniaManipulatora = 0 THEN  //Lavá M6 - 4F
						P2_Srobovanie.PAR.RR_TypModelu:= '4F';
						P2_Srobovanie.STAV.RR_Polohovanie_BUSY:= TRUE;
						P2_Srobovanie.CMD.RR_PolohujManipulator:= FALSE;
						SC_P2_Srobovanie.ResetStep:= TRUE;
						SC_P2_Srobovanie.Step:= 110;
					ELSIF P2_Srobovanie.PAR.RR_IndexPolohovaniaManipulatora = 1 THEN  //Pravá M6 - 4F
						P2_Srobovanie.PAR.RR_TypModelu:= '4F';
						P2_Srobovanie.STAV.RR_Polohovanie_BUSY:= TRUE;
						P2_Srobovanie.CMD.RR_PolohujManipulator:= FALSE;
						SC_P2_Srobovanie.ResetStep:= TRUE;
						SC_P2_Srobovanie.Step:= 130;
					ELSIF P2_Srobovanie.PAR.RR_IndexPolohovaniaManipulatora = 2 THEN  //Lavá M4 - 4F
						P2_Srobovanie.PAR.RR_TypModelu:= '4F';
						P2_Srobovanie.STAV.RR_Polohovanie_BUSY:= TRUE;
						P2_Srobovanie.CMD.RR_PolohujManipulator:= FALSE;
						SC_P2_Srobovanie.ResetStep:= TRUE;
						SC_P2_Srobovanie.Step:= 160;
					ELSIF P2_Srobovanie.PAR.RR_IndexPolohovaniaManipulatora = 3 THEN  //Pravá M4 - 4F
						P2_Srobovanie.PAR.RR_TypModelu:= '4F';
						P2_Srobovanie.STAV.RR_Polohovanie_BUSY:= TRUE;
						P2_Srobovanie.CMD.RR_PolohujManipulator:= FALSE;
						SC_P2_Srobovanie.ResetStep:= TRUE;
						SC_P2_Srobovanie.Step:= 180;
					ELSIF P2_Srobovanie.PAR.RR_IndexPolohovaniaManipulatora = 4 THEN  //Lavá M6 - 5F
						P2_Srobovanie.PAR.RR_TypModelu:= '5F';
						P2_Srobovanie.STAV.RR_Polohovanie_BUSY:= TRUE;
						P2_Srobovanie.CMD.RR_PolohujManipulator:= FALSE;
						SC_P2_Srobovanie.ResetStep:= TRUE;
						SC_P2_Srobovanie.Step:= 110;
					ELSIF P2_Srobovanie.PAR.RR_IndexPolohovaniaManipulatora = 5 THEN  //Pravá M6 - 5F
						P2_Srobovanie.PAR.RR_TypModelu:= '5F';
						P2_Srobovanie.CMD.RR_PolohujManipulator:= FALSE;
						P2_Srobovanie.STAV.RR_Polohovanie_BUSY:= TRUE;
						SC_P2_Srobovanie.ResetStep:= TRUE;
						SC_P2_Srobovanie.Step:= 130;
					ELSIF P2_Srobovanie.PAR.RR_IndexPolohovaniaManipulatora = 6 THEN  //Lavá M4 - 5F
						P2_Srobovanie.PAR.RR_TypModelu:= '5F';
						P2_Srobovanie.STAV.RR_Polohovanie_BUSY:= TRUE;
						P2_Srobovanie.CMD.RR_PolohujManipulator:= FALSE;
						SC_P2_Srobovanie.ResetStep:= TRUE;
						SC_P2_Srobovanie.Step:= 160;
					ELSIF P2_Srobovanie.PAR.RR_IndexPolohovaniaManipulatora = 7 THEN  //Pravá M4 - 5F
						P2_Srobovanie.PAR.RR_TypModelu:= '5F';
						P2_Srobovanie.STAV.RR_Polohovanie_BUSY:= TRUE;
						P2_Srobovanie.CMD.RR_PolohujManipulator:= FALSE;
						SC_P2_Srobovanie.ResetStep:= TRUE;
						SC_P2_Srobovanie.Step:= 180;
					ELSIF P2_Srobovanie.PAR.RR_IndexPolohovaniaManipulatora = 8 THEN  //Lavá M5 - 5H
						P2_Srobovanie.STAV.RR_Polohovanie_BUSY:= TRUE;
						P2_Srobovanie.CMD.RR_PolohujManipulator:= FALSE;
						SC_P2_Srobovanie.ResetStep:= TRUE;
						SC_P2_Srobovanie.Step:= 200;
					ELSIF P2_Srobovanie.PAR.RR_IndexPolohovaniaManipulatora = 9 THEN  //Pravá M5 - 5H
						P2_Srobovanie.STAV.RR_Polohovanie_BUSY:= TRUE;
						P2_Srobovanie.CMD.RR_PolohujManipulator:= FALSE;
						SC_P2_Srobovanie.ResetStep:= TRUE;
						SC_P2_Srobovanie.Step:= 220;
					ELSIF P2_Srobovanie.PAR.RR_IndexPolohovaniaManipulatora = 10 THEN  //Stredná M4 - 5H
						P2_Srobovanie.STAV.RR_Polohovanie_BUSY:= TRUE;
						P2_Srobovanie.CMD.RR_PolohujManipulator:= FALSE;
						SC_P2_Srobovanie.ResetStep:= TRUE;
						SC_P2_Srobovanie.Step:= 250;
					ELSIF P2_Srobovanie.PAR.RR_IndexPolohovaniaManipulatora = 11 THEN  //Pozicia odobratia skrutky M4
						P2_Srobovanie.STAV.RR_Polohovanie_BUSY:= TRUE;
						P2_Srobovanie.CMD.RR_PolohujManipulator:= FALSE;
						SC_P2_Srobovanie.ResetStep:= TRUE;
						SC_P2_Srobovanie.Step:= 440;
					END_IF
				END_IF
				P2_Srobovanie.CMD.RR_PolohujManipulator:= FALSE;
			END_IF

	END_CASE

				END_PROGRAM

PROGRAM _EXIT
				(* Insert code here *)

				END_PROGRAM
```

#### Variables.var - Local variables
```iecst
VAR
	FazaNavratu : UINT := 0;
	CasSrobovania : REAL := 0.0;
	PocetCisteniSkrutkovacky : USINT := 0;
	M6_PrevodMomentu : PrevodMomentu;
	M4_PrevodMomentu : PrevodMomentu;
	M5_PrevodMomentu : PrevodMomentu;
	CasEnable_1 : TON;
	CasEnable_2 : TON;
	CasEnable_3 : TON := (0);
	CasResetServo_1 : TON;
	CasResetServo_2 : TON;
	CasResetServo_3 : TON;
	SC_SkrutkovaciSet_M6 : SequenceControlTyp := (0);
	SC_SkrutkovaciSet_M4 : SequenceControlTyp := (0);
	SC_SkrutkovaciSet_M5 : SequenceControlTyp := (0);
END_VAR
```
